# EPICS substitutions: src/iocdoc/testfiles/iocBoot/ioc495idc/templates/dac128V.substitutions
file "$(DAC128V)/dac128VApp/Db/singleDAC.db"
{pattern
{P,      D, N, S, PORT,   EGUL,  EGUF, DRVL, DRVH, LOPR, HOPR, PREC,     LINR, VAL}
{495idc:, 1, 1, 0, DAC1,    -10,    10, -10,  10,   -10,  10,   3,    "LINEAR", 0}
{495idc:, 1, 2, 1, DAC1,    -10,    10, -10,  10,   -10,  10,   3,    "LINEAR", 0}
{495idc:, 1, 3, 2, DAC1,    -10,    10, -10,  10,   -10,  10,   3,    "LINEAR", 0}
{495idc:, 1, 4, 3, DAC1,    -10,    10, -10,  10,   -10,  10,   3,    "LINEAR", 0}
{495idc:, 1, 5, 4, DAC1,    -10,    10, -10,  10,   -10,  10,   3,    "LINEAR", 0}
{495idc:, 1, 6, 5, DAC1,    -10,    10, -10,  10,   -10,  10,   3,    "LINEAR", 0}
{495idc:, 1, 7, 6, DAC1,    -10,    10, -10,  10,   -10,  10,   3,    "LINEAR", 0}
{495idc:, 1, 8, 7, DAC1,    -10,    10, -10,  10,   -10,  10,   3,    "LINEAR", 0}
# Channel 2 is in volts, -10 to 10, but only allow driving 0 to 10
#! {495idc:, 1, 2, 1, DAC1,    -10,    10,   0,  10,     0,  10,   3,    "LINEAR", 0}
}
